(* IEC 61131-3 sources: test/Class/_LimitMin, 1 file *)

(* ---- _LimitMin.st ---- *)
#ifndef OS_STARTVERSION_SALAMANDER
#define OS_STARTVERSION_SALAMANDER  16#09000
#endif

// date Limit for Salamander-OS
#define MINDATE_SALAMANDER_YEAR     2010
#define MINDATE_SALAMANDER_MONTH    1
#define MINDATE_SALAMANDER_DAY      1

// date Limit for RtOS
#define MINDATE_RTOS_YEAR     1990
#define MINDATE_RTOS_MONTH    1
#define MINDATE_RTOS_DAY      1

(*!
<Class
	Name               = "_LimitMin"
	Revision           = "0.2"
	RealtimeTask       = "false"
	CyclicTask         = "false"
	BackgroundTask     = "false"
	Sigmatek           = "true"
	OSInterface        = "false"
	HighPriority       = "false"
	Automatic          = "false"
	UpdateMode         = "Prescan"
	SharedCommandTable = "true"
	Objectsize         = "(284,120)"
	Comment            = "is used to display lower limit of server">
	<Channels>
		<Server
			Name           = "Server0"
			Initialize     = "false"
			Visualized     = "true"
			WriteProtected = "true">
		</Server>
	</Channels>
	<RevDoku>
		<Owner/>
		<Dokumentation Revision="0.2" Date="2016-10-20" Author="HubChr" Company="Sigmatek" Description="-) Class showed the same values for Rtos and Salamander (Maximum Date on Salamander is different!)"/>
	</RevDoku>
	<Network Name="_LimitMin">
		<!-- List of Components in this network -->
		<Components>
			<Object
				Name       = "_base"
				Class      = "_MyIO"
				Position   = "(270,150)"
				Visualized = "true">
				<Channels>
					<Server Name="Refresh"/>
					<Server Name="Server0"/>
					<Client Name="Graphic"/>
					<Client Name="Lse"/>
				</Channels>
			</Object>
		</Components>
		<Comments>
		</Comments>
		<!-- List of Connections in this network -->
		<Connections>
			<Connection Source="this.Server0" Destination="_base.Server0" Vertices="(742,210),(570,240),"/>
			<Connection Source="_base.Lse" Destination="this.Lse" Vertices="(270,240),(38,210),"/>
		</Connections>
		<!-- Headerfiles -->
		<Options>
		</Options>
	</Network>
</Class>
*)
#pragma using _MyIO

_LimitMin : CLASS
: _MyIO
  //Servers:
  //Clients:
  //Variables:
  //Functions:
				//! <Function Comment="[#ENGLISH]&#13;&#10;this method is called everytime when system wants to redraw the io&#13;&#10;&#13;&#10;pio ....... pointer to io information&#13;&#10;pr ........ pointer to result information&#13;&#10;pv ........ pointer to io variableinformation&#13;&#10;input ..... TRUE it&apos;s an input / FALSE it&apos;s an output&#13;&#10;&#13;&#10;for the returnstatement there are 3 different possibilities&#13;&#10;_IDLE ..... the system should goon like it is (system goes on)&#13;&#10;_IDIDIT ... i did it (system is ready)&#13;&#10;_IFAILED .. i tried to do my best, but i failed (system is ready)&#13;&#10;&#13;&#10;if you want to draw the io let&apos;s return _IDIDIT&#13;&#10;" Name="Draw"/>
	FUNCTION __CDECL VIRTUAL GLOBAL Draw
		VAR_INPUT
			pio 	: ^_IO;			//! <Variable Comment="pointer to _IO information" Name="Draw.pio"/>
			pr 	: ^_RESULT;			//! <Variable Comment="pointer to _RESULT information" Name="Draw.pr"/>
			pv 	: ^_VARIABLE;			//! <Variable Comment="pointer to io _VARIABLE information" Name="Draw.pv"/>
			input 	: BOOL;			//! <Variable Comment="TRUE it&apos;s an input&#13;&#10;FALSE it&apos;s an output" Name="Draw.input"/>
		END_VAR
		VAR_OUTPUT
			retcode (EAX) 	: _DOIT;			//! <Variable Comment="for the returnstatement there are 3 different possibilities&#13;&#10;  _IDLE ..... the system should goon like it is (system goes on)&#13;&#10;  _IDIDIT ... i did it (system is ready)&#13;&#10;  _IFAILED .. i tried to do my best, but i failed (system is re" Name="Draw.retcode"/>
		END_VAR;
				//! <Function Comment="[#ENGLISH]&#13;&#10;this method is called everytime when system wants to get data for defined io.&#13;&#10;&#13;&#10;pr ........ pointer to result information&#13;&#10;pio ....... pointer to io information&#13;&#10;pv ........ pointer to io variableinformation&#13;&#10;input ..... _TRUE it&apos;s an input / _FALSE it&apos;s an output&#13;&#10;&#13;&#10;for the returnstatement there are 3 different possibilities&#13;&#10;_IDLE ..... the system should goon like it is (system goes on)&#13;&#10;_IDIDIT ... i did it (system is ready)&#13;&#10;_IFAILED .. i tried to do my best, but i failed (system is ready)&#13;&#10;&#13;&#10;if you want to do it let&apos;s return _IDIDIT and initialize the  structure _RESULT&#13;&#10;" Name="GetData"/>
	FUNCTION __CDECL VIRTUAL GLOBAL GetData
		VAR_INPUT
			pr 	: ^_RESULT;			//! <Variable Comment="pointer to _RESULT information" Name="GetData.pr"/>
			pio 	: ^_IO;			//! <Variable Comment="pointer to _IO information" Name="GetData.pio"/>
			pv 	: ^_VARIABLE;			//! <Variable Comment="pointer to _VARIABLE information given by LSE" Name="GetData.pv"/>
			input 	: BOOL;			//! <Variable Comment="TRUE it&apos;s an input&#13;&#10;FALSE it&apos;s an output" Name="GetData.input"/>
		END_VAR
		VAR_OUTPUT
			retcode (EAX) 	: _DOIT;			//! <Variable Comment="for the returnstatement there are 3 different possibilities&#13;&#10;  _IDLE ..... the system should goon like it is (system goes on)&#13;&#10;  _IDIDIT ... i did it (system is ready)&#13;&#10;  _IFAILED .. i tried to do my best, but i failed (system is ready)" Name="GetData.retcode"/>
		END_VAR;
  //Tables:
	FUNCTION @STD
		VAR_OUTPUT
			ret_code	: CONFSTATES;
		END_VAR;
	FUNCTION GLOBAL TAB @CT_;
END_CLASS;

#pragma using _Lse

//*********************Inserted from .\_LimitMin\_LimitMin_00_00.st*********************

#pragma warning (disable: 73)
//[#ENGLISH]
//this method is called everytime when system wants to get data for defined io.
//
//pr ........ pointer to result information
//pio ....... pointer to io information
//pv ........ pointer to io variableinformation
//input ..... _TRUE it's an input / _FALSE it's an output
//
//for the returnstatement there are 3 different possibilities
//_IDLE ..... the system should goon like it is (system goes on)
//_IDIDIT ... i did it (system is ready)
//_IFAILED .. i tried to do my best, but i failed (system is ready)
//
//if you want to do it let's return _IDIDIT and initialize the  structure _RESULT

FUNCTION __CDECL VIRTUAL GLOBAL _LimitMin::GetData
VAR_INPUT
	pr		: ^_RESULT;
	pio		: ^_IO;
	pv		: ^_VARIABLE;
	input		: BOOL;
END_VAR
VAR_OUTPUT
	retcode		: _DOIT;
END_VAR

  pr^.value := pr^.rmin;
  retcode   := _IDLE;

END_FUNCTION //__CDECL VIRTUAL GLOBAL _LimitMin::GetData

FUNCTION __CDECL VIRTUAL GLOBAL _LimitMin::Draw
	VAR_INPUT
		pio 	: ^_IO;
		pr 	: ^_RESULT;
		pv 	: ^_VARIABLE;
		input 	: BOOL;
	END_VAR
	VAR_OUTPUT
		retcode (EAX) 	: _DOIT;
	END_VAR
  VAR
  	txt : array[0..39] of _CHAR;
    tim : _TIME;
    dat : _DATE;
    format : uint;
  END_VAR

  retcode := _IDLE;

  if(pv^.info.vartype = FTIME) then
    tim.hour := 0;
    tim.minute := 0;
    tim.second := 0;
    format_time(#txt[0], #tim, pv^.info.format);
    OutMultiTextAlign(#txt[0], 0, #pio^.space, pio^.font, pio^.attrib, pio^.frametype, pio^.coltxt, pio^.colback, pio^.colframe, sizeof(_CHAR));
    retcode := _IDIDIT;
  elsif(pv^.info.vartype = FDATE) then

    // -- HubChr v0.2 Maximum Date depends on platform!
    if _rtosversion >= OS_STARTVERSION_SALAMANDER then
      dat.year := MINDATE_SALAMANDER_YEAR;
      dat.month := MINDATE_SALAMANDER_MONTH;
      dat.day := MINDATE_SALAMANDER_DAY;
    else
      dat.year := MINDATE_RTOS_YEAR;
      dat.month := MINDATE_RTOS_MONTH;
      dat.day := MINDATE_RTOS_DAY;
    end_if;
    // -- End HubChr v0.2

    format := pv^.info.format;
    case format of
      SIZE_DDMMYY : dat.year := 1990;
      SIZE_WWDDMM : format := SIZE_DDMM;
      SIZE_WWDDMMYYYY : format := SIZE_DDMMYYYY;
    end_case;

    format_date(#txt[0], #dat, format);
    OutMultiTextAlign(#txt[0], 0, #pio^.space, pio^.font, pio^.attrib, pio^.frametype, pio^.coltxt, pio^.colback, pio^.colframe, sizeof(_CHAR));
    retcode := _IDIDIT;
  end_if;

END_FUNCTION
